// TIA Portal V17 export
// export: Created 2024-08-07T21:44:16.479987Z, ExportSetting WithDefaults, DisplayName Totally Integrated Automation Portal, DisplayVersion V17 Update 7, DisplayName TIA Portal Openness, DisplayVersion V17 Update 7, DisplayName TIA Portal Version Control Interface, DisplayVersion V17, DisplayName SINAMICS Startdrive Advanced, DisplayVersion V17 SP2, DisplayName SINAMICS Startdrive G110M, G120, G120C, G120D, G120P, G115D, DisplayVersion V17 SP2, DisplayName SINAMICS Startdrive G130, G150, S120, S150, SINAMICS MV, S210, DisplayVersion V17 SP2, DisplayName STEP 7 Professional, DisplayVersion V17 Update 7, DisplayName STEP 7 Safety, DisplayVersion V17 Update 6, DisplayName WinCC Advanced / Unified PC, DisplayVersion V17 Update 7
TYPE "methodListType"
// stored: IsFailsafeCompliant false
   STRUCT
      MethodCount { ExternalAccessible := 'False'; ExternalVisible := 'False'; ExternalWritable := 'False'} : UInt;
      ObjectNodes { ExternalAccessible := 'False'; ExternalVisible := 'False'; ExternalWritable := 'False'; S7_SetPoint := 'True'} : Array[0..0] of OPC_UA_NodeId;
      MethodNodes { ExternalAccessible := 'False'; ExternalVisible := 'False'; ExternalWritable := 'False'; S7_SetPoint := 'True'} : Array[0..0] of OPC_UA_NodeId;
      MethodHdls { ExternalAccessible := 'False'; ExternalVisible := 'False'; ExternalWritable := 'False'} : Array[0..0] of DWord;
   END_STRUCT;
   // ObjectNodes[0].NamespaceIndex := 0;
   // ObjectNodes[0].Identifier := WSTRING#'"OPCMethodSetMachineTime_DB"';
   // ObjectNodes[0].IdentifierType := 1;
   // MethodNodes[0].NamespaceIndex := 0;
   // MethodNodes[0].Identifier := WSTRING#'"OPCMethodSetMachineTime_DB".Method';
   // MethodNodes[0].IdentifierType := 1;
END_TYPE
